FUNCTION_BLOCK POU
VAR_INPUT
END_VAR
VAR_OUTPUT
END_VAR
VAR
END_VAR

END_FUNCTION_BLOCK

(* stored: Version 1.1.0.1
   POU POU: Id {9d4b132c-1e39-4fc2-8b2e-92e2d990dbcd}, SpecialFunc None *)
